PROGRAM InputPositionProtection
VAR
END_VAR

(************Input Position Protection****************)
IF Axis1_TargetPosition_retain>=Axis1_minPosition AND Axis1_TargetPosition_retain<=Axis1_maxPosition THEN
	Axis1_InputPositionOutOfRange:=FALSE;
ELSE
	Axis1_InputPositionOutOfRange:=TRUE;
END_IF
IF Axis2_TargetPosition_retain>=Axis2_minPosition AND Axis2_TargetPosition_retain<=Axis2_maxPosition THEN
	Axis2_InputPositionOutOfRange:=FALSE;
ELSE
	Axis2_InputPositionOutOfRange:=TRUE;
END_IF

END_PROGRAM

(* stored: Version 1.1.0.1, ProductVersion 3.1.4024.6
   POU InputPositionProtection: Id {d08ef58f-fced-4486-b224-0df6caf71e1d}, SpecialFunc None *)
